// Mitsubishi GX Works2 project: Group29   PLC: FX3G

// global labels: Global1
VAR_GLOBAL
  emergency AT X005 : BOOL;
  low_stock AT M2 : BOOL;
  light7 AT Y007 : BOOL;
  start_work_day AT X007 : BOOL;
  switch1 AT X001 : BOOL;
  inputAnalog AT D8280 : INT;
  outputAnalog AT D1400 : REAL;
END_VAR
VAR_GLOBAL CONSTANT
  const400 : REAL := 400;
  const5 : REAL := 5;
END_VAR
VAR_GLOBAL
  lightPinuk AT M5 : BOOL;
  lightRegular AT M7 : BOOL;
  input_raspberry AT D1100 : REAL;
  raspberry_stock AT D1200 : REAL;
  input_lemon AT D1103 : REAL;
  lemon_stock AT D1203 : REAL;
  input_stabilizer AT D1106 : REAL;
  stabilizer_stock AT D1206 : REAL;
  input_gummies AT D1109 : REAL;
  gummy_stock AT D1209 : REAL;
END_VAR
VAR_GLOBAL CONSTANT
  packages_start : REAL;
END_VAR
VAR_GLOBAL
  packges_regular AT D1212 : REAL;
  low_stock_stop AT M2 : BOOL;
  switchPinuk AT M5 : BOOL;
END_VAR
VAR_GLOBAL CONSTANT
  const6 : REAL := 6;
END_VAR
VAR_GLOBAL
  switchRegular AT M7 : BOOL;
  notInRange AT M9 : BOOL;
  switchNotInRange AT M9 : BOOL;
END_VAR
VAR_GLOBAL CONSTANT
  constantAmountRasperry1 : REAL := 385;
  constantAmountLemon1 : REAL := 665;
  constantAmountStabilzer1 : REAL := 210;
  constantAmountGummy1 : REAL := 70;
END_VAR
VAR_GLOBAL
  enoughRaspberry1 AT M20 : BOOL;
  enoughLemon1 AT M23 : BOOL;
  enoughStabilizer1 AT M26 : BOOL;
  emnoghGummy AT M29 : BOOL;
  emnoghGummy1 AT M29 : BOOL;
END_VAR
VAR_GLOBAL CONSTANT
  constantAmountRasperry2 : REAL := 280;
  constantAmountLemon2 : REAL := 455;
  constantAmountStabilzer2 : REAL := 105;
  constantAmountGummy2 : REAL := 28;
END_VAR
VAR_GLOBAL
  enoughRaspberry2 AT M32 : BOOL;
  enoughLemon2 AT M35 : BOOL;
  enoughStabilizer2 AT M38 : BOOL;
  emnoghGummy2 AT M41 : BOOL;
  fullStock AT M44 : BOOL;
  switchFullStock AT M44 : BOOL;
  lightLowStock AT M2 : BOOL;
  packges_pinuk AT D1215 : REAL;
END_VAR
VAR_GLOBAL CONSTANT
  conatant1 : REAL := 1.0;
END_VAR
VAR_GLOBAL
  Light5Sec AT M70 : BOOL;
  TStimer50 AT TS50 : BOOL;
  Timer5sec AT TC50 : BOOL;
  switch5Sec AT M70 : BOOL;
  switch2 AT X002 : BOOL;
  TStimer80 AT TS80 : BOOL;
  switch3 AT X003 : BOOL;
  LightCooling AT M73 : BOOL;
  switchCooling AT M73 : BOOL;
END_VAR
VAR_GLOBAL CONSTANT
  const80 : REAL := 80;
  const100 : REAL := 100;
  const50 : REAL := 50;
  const70 : REAL := 70;
END_VAR
VAR_GLOBAL
  Timer50 AT TC50 : BOOL;
END_VAR
VAR_GLOBAL CONSTANT
  timer50TV : INT := 50;
END_VAR
VAR_GLOBAL
  Timer80 AT TC80 : BOOL;
END_VAR
VAR_GLOBAL CONSTANT
  timer80TV : INT := 80;
END_VAR
VAR_GLOBAL
  switch7 AT Y007 : BOOL;
  raspberry_cooling_regular AT D1220 : REAL;
  lemon_cooling_regular AT D1223 : REAL;
  raspberry_cooling_pinuk AT D1226 : REAL;
  lemon_cooling_pinuk AT D1229 : REAL;
  Light0 AT Y000 : BOOL;
  Light2 AT Y002 : BOOL;
  raspberry_cooling AT D1226 : REAL;
  lemon_cooling AT D1229 : REAL;
  total_add_raspberry AT D1232 : REAL;
  total_add_lemon AT D1235 : REAL;
  switch0 AT Y000 : BOOL;
  switchMix AT M86 : BOOL;
  mixHelp AT M76 : BOOL;
  Timer5 AT TC5 : BOOL;
END_VAR
VAR_GLOBAL CONSTANT
  const20 : INT := 1;
  const1timer : INT := 1;
END_VAR
VAR_GLOBAL
  TStimer5 AT TS5 : BOOL;
END_VAR
VAR_GLOBAL CONSTANT
  const10timer : INT := 5;
END_VAR
VAR_GLOBAL
  Light5 AT Y005 : BOOL;
  Timer6 AT TC6 : BOOL;
  TStimer6 AT TS6 : BOOL;
  Light6 AT Y006 : BOOL;
  switch5 AT Y005 : BOOL;
  switch6 AT Y006 : BOOL;
  regularCounter AT CC3 : BOOL;
END_VAR
VAR_GLOBAL CONSTANT
  const3 : INT := 3;
END_VAR
VAR_GLOBAL
  outConterRegular AT CS3 : BOOL;
  storage AT D1240 : REAL;
END_VAR
VAR_GLOBAL CONSTANT
  const0 : REAL;
END_VAR
VAR_GLOBAL
  isPinuk AT M79 : BOOL;
  isRegular AT M82 : BOOL;
  LightMix AT M86 : BOOL;
  switchFinishCooling AT Y002 : BOOL;
  light2TurnedOff AT M98 : BOOL;
  MixTimerPinuk AT TC1 : BOOL;
  MixTimerregular AT TC2 : BOOL;
END_VAR
VAR_GLOBAL CONSTANT
  PinukMixDuration : INT := 50;
  RegularMixDuration : INT := 30;
END_VAR
VAR_GLOBAL
  TSRegular AT TS2 : BOOL;
  TSPinuk AT TS1 : BOOL;
END_VAR
VAR_GLOBAL CONSTANT
  const1time5 : INT := 1;
  const5timer : INT := 5;
END_VAR
VAR_GLOBAL
  finishCooling AT M99 : BOOL;
  mAor AT M90 : BOOL;
  finishMix AT M96 : BOOL;
  LightStartMix AT M86 : BOOL;
  switchStartMix AT M86 : BOOL;
  storage_out AT D1280 : REAL;
END_VAR
VAR_GLOBAL CONSTANT
  const40 : REAL := 40;
END_VAR
VAR_GLOBAL
  OUTPUT AT D8282 : DINT;
END_VAR
VAR_GLOBAL CONSTANT
  const350 : REAL := 350;
  const560 : REAL := 560;
  const700 : REAL := 700;
  const490 : REAL := 490;
END_VAR
VAR_GLOBAL
  total_respberry_lemon_pinuk AT D1260 : REAL;
  total_ice_pinuk AT D1260 : REAL;
  Mixing_container AT D1260 : REAL;
  raspberry_cooling_container AT D1226 : REAL;
  lemon_cooling_container AT D1229 : REAL;
END_VAR

// task Task_01 (event TRUE, interval 0, priority 31): POU_01

PROGRAM POU_01
(* structured ladder/FBD written out as ST: instructions are called as NAME(EN, inputs, outputs); _pN, _eN, _tN stand for wires *)
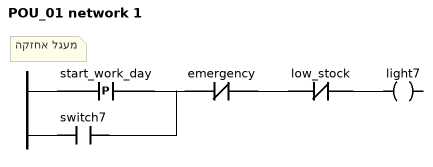
(* network 1 *)
(* מעגל אחזקה *)
light7 := ((LDP(TRUE, start_work_day) OR switch7) AND NOT emergency) AND NOT low_stock;
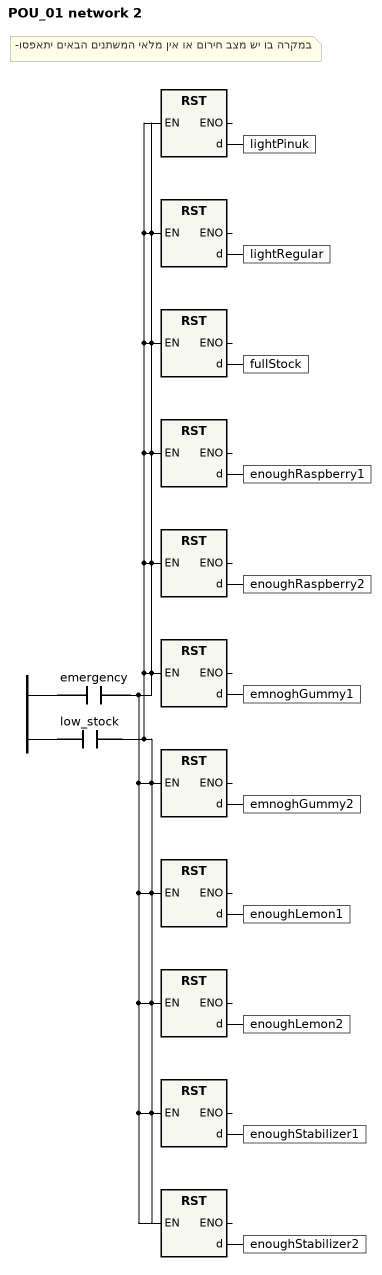
(* network 2 *)
(* במקרה בו יש מצב חירום או אין מלאי המשתנים הבאים יתאפסו- *)
_p1 := emergency OR low_stock;
RST(_p1, lightPinuk);
RST(_p1, lightRegular);
RST(_p1, fullStock);
RST(_p1, enoughRaspberry1);
RST(_p1, enoughRaspberry2);
RST(_p1, emnoghGummy1);
RST(_p1, emnoghGummy2);
RST(_p1, enoughLemon1);
RST(_p1, enoughLemon2);
RST(_p1, enoughStabilizer1);
RST(_p1, enoughStabilizer2);
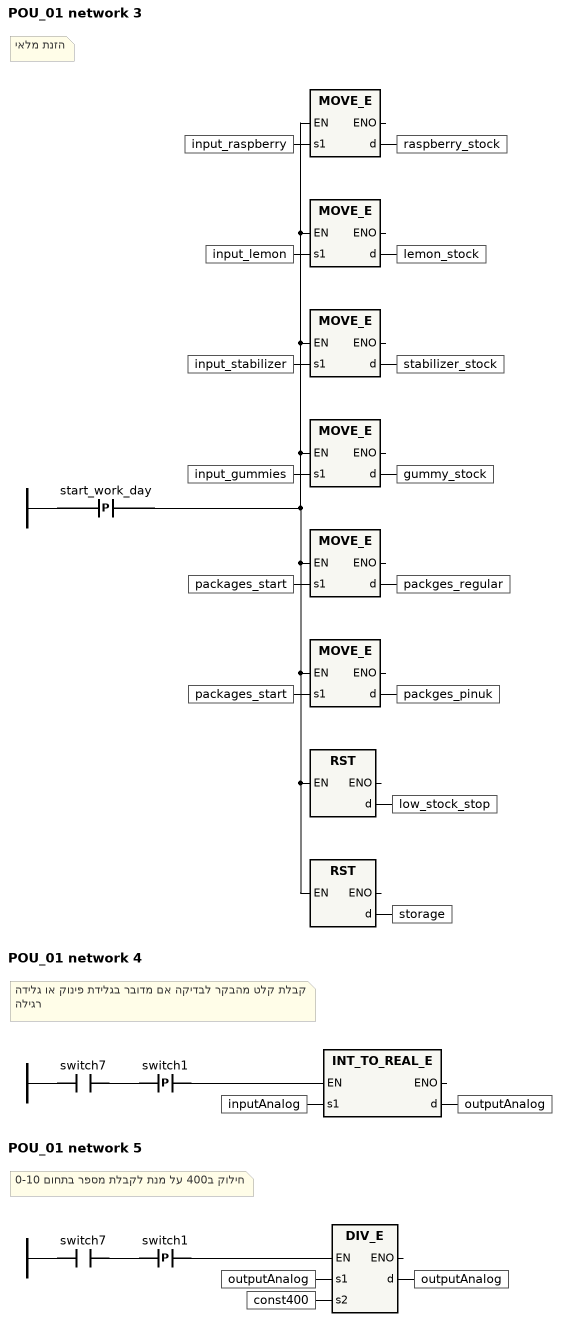
(* network 3 *)
(* הזנת מלאי *)
_p1 := LDP(TRUE, start_work_day);
MOVE_E(_p1, input_raspberry, raspberry_stock);
MOVE_E(_p1, input_lemon, lemon_stock);
MOVE_E(_p1, input_stabilizer, stabilizer_stock);
MOVE_E(_p1, input_gummies, gummy_stock);
MOVE_E(_p1, packages_start, packges_regular);
MOVE_E(_p1, packages_start, packges_pinuk);
RST(_p1, low_stock_stop);
RST(_p1, storage);
(* network 4 *)
(* קבלת קלט מהבקר לבדיקה אם מדובר בגלידת פינוק או גלידה רגילה *)
INT_TO_REAL_E(switch7 AND LDP(TRUE, switch1), inputAnalog, outputAnalog);
(* network 5 *)
(* חילוק ב400 על מנת לקבלת מספר בתחום 0-10 *)
DIV_E(switch7 AND LDP(TRUE, switch1), outputAnalog, const400, outputAnalog);
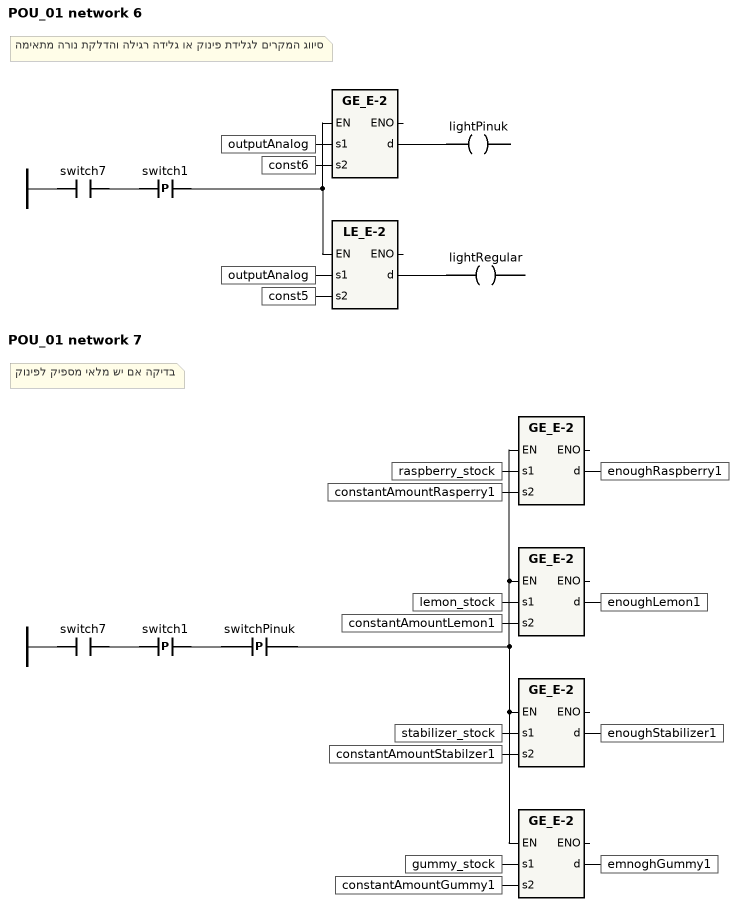
(* network 6 *)
(* סיווג המקרים לגלידת פינוק או גלידה רגילה והדלקת נורה מתאימה *)
_p1 := switch7 AND LDP(TRUE, switch1);
GE_E(_p1, outputAnalog, const6, _t2);
lightPinuk := _t2;
LE_E(_p1, outputAnalog, const5, _t3);
lightRegular := _t3;
(* network 7 *)
(* בדיקה אם יש מלאי מספיק לפינוק *)
_p1 := switch7 AND LDP(TRUE, switch1) AND LDP(TRUE, switchPinuk);
GE_E(_p1, raspberry_stock, constantAmountRasperry1, enoughRaspberry1);
GE_E(_p1, lemon_stock, constantAmountLemon1, enoughLemon1);
GE_E(_p1, stabilizer_stock, constantAmountStabilzer1, enoughStabilizer1);
GE_E(_p1, gummy_stock, constantAmountGummy1, emnoghGummy1);
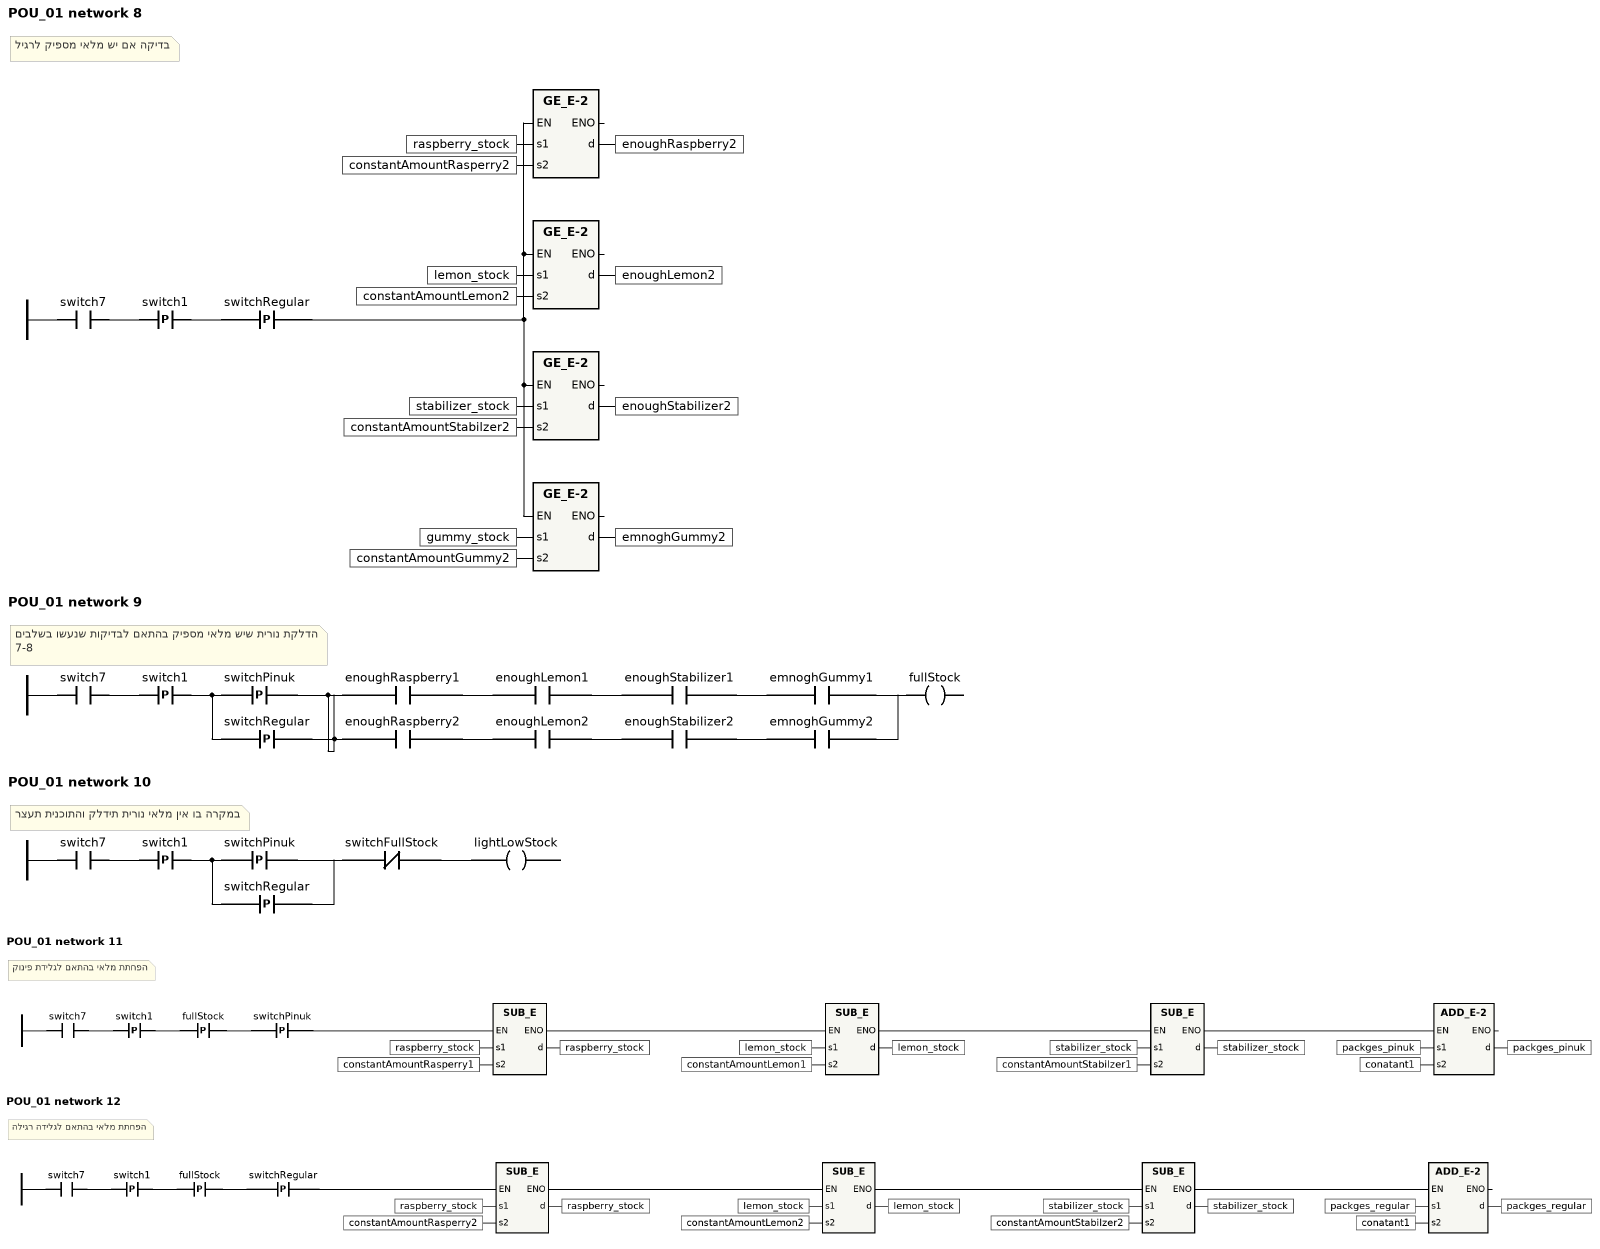
(* network 8 *)
(* בדיקה אם יש מלאי מספיק לרגיל *)
_p1 := switch7 AND LDP(TRUE, switch1) AND LDP(TRUE, switchRegular);
GE_E(_p1, raspberry_stock, constantAmountRasperry2, enoughRaspberry2);
GE_E(_p1, lemon_stock, constantAmountLemon2, enoughLemon2);
GE_E(_p1, stabilizer_stock, constantAmountStabilzer2, enoughStabilizer2);
GE_E(_p1, gummy_stock, constantAmountGummy2, emnoghGummy2);
(* network 9 *)
(* הדלקת נורית שיש מלאי מספיק בהתאם לבדיקות שנעשו בשלבים 7-8 *)
_p1 := switch7 AND LDP(TRUE, switch1);
_p2 := (_p1 AND LDP(TRUE, switchPinuk)) OR (_p1 AND LDP(TRUE, switchRegular));
fullStock := (_p2 AND enoughRaspberry1 AND enoughLemon1 AND enoughStabilizer1 AND emnoghGummy1) OR (_p2 AND enoughRaspberry2 AND enoughLemon2 AND enoughStabilizer2 AND emnoghGummy2);
(* network 10 *)
(* במקרה בו אין מלאי נורית תידלק והתוכנית תעצר *)
_p1 := switch7 AND LDP(TRUE, switch1);
lightLowStock := ((_p1 AND LDP(TRUE, switchPinuk)) OR (_p1 AND LDP(TRUE, switchRegular))) AND NOT switchFullStock;
(* network 11 *)
(* הפחתת מלאי בהתאם לגלידת פינוק *)
_e1 := SUB_E(switch7 AND LDP(TRUE, switch1) AND LDP(TRUE, fullStock) AND LDP(TRUE, switchPinuk), raspberry_stock, constantAmountRasperry1, raspberry_stock);
_e2 := SUB_E(_e1, lemon_stock, constantAmountLemon1, lemon_stock);
_e3 := SUB_E(_e2, stabilizer_stock, constantAmountStabilzer1, stabilizer_stock);
ADD_E(_e3, packges_pinuk, conatant1, packges_pinuk);
(* network 12 *)
(* הפחתת מלאי בהתאם לגלידה רגילה *)
_e1 := SUB_E(switch7 AND LDP(TRUE, switch1) AND LDP(TRUE, fullStock) AND LDP(TRUE, switchRegular), raspberry_stock, constantAmountRasperry2, raspberry_stock);
_e2 := SUB_E(_e1, lemon_stock, constantAmountLemon2, lemon_stock);
_e3 := SUB_E(_e2, stabilizer_stock, constantAmountStabilzer2, stabilizer_stock);
ADD_E(_e3, packges_regular, conatant1, packges_regular);
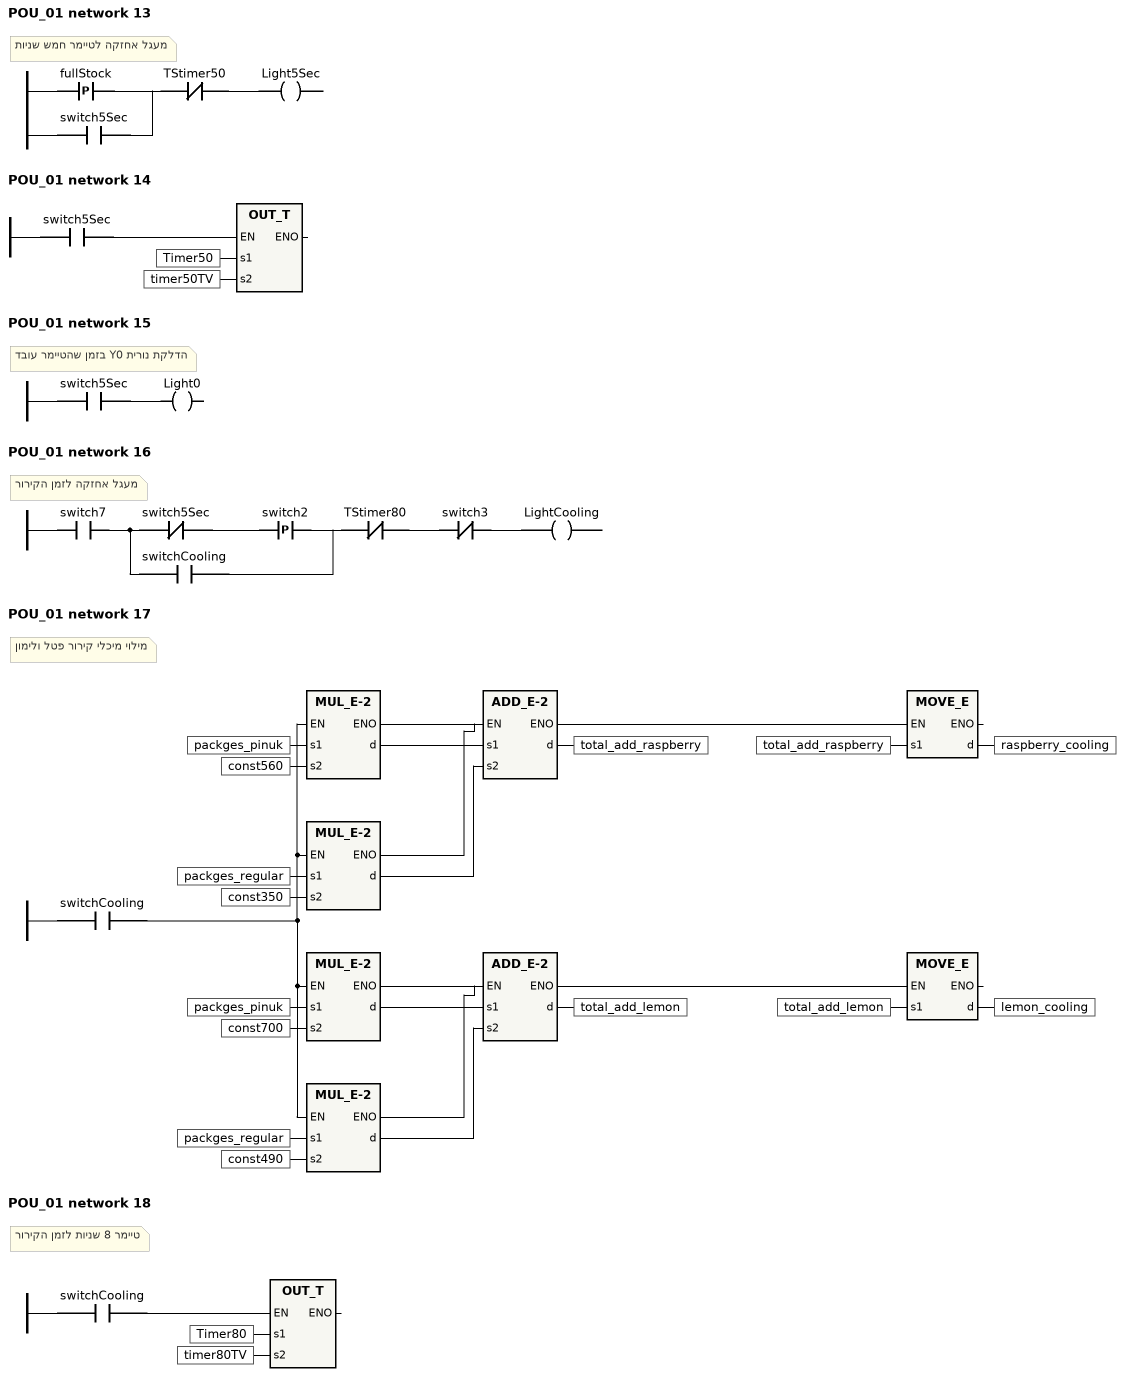
(* network 13 *)
(* מעגל אחזקה לטיימר חמש שניות *)
Light5Sec := (LDP(TRUE, fullStock) OR switch5Sec) AND NOT TStimer50;
(* network 14 *)
OUT_T(switch5Sec, Timer50, timer50TV);
(* network 15 *)
(* הדלקת נורית Y0 בזמן שהטיימר עובד *)
Light0 := switch5Sec;
(* network 16 *)
(* מעגל אחזקה לזמן הקירור *)
LightCooling := (((switch7 AND NOT switch5Sec AND LDP(TRUE, switch2)) OR (switch7 AND switchCooling)) AND NOT TStimer80) AND NOT switch3;
(* network 17 *)
(* מילוי מיכלי קירור פטל ולימון *)
_e2 := MUL_E(switchCooling, packges_pinuk, const560, _t1);
_e4 := MUL_E(switchCooling, packges_regular, const350, _t3);
_e5 := ADD_E(_e2 OR _e4, _t1, _t3, total_add_raspberry);
MOVE_E(_e5, total_add_raspberry, raspberry_cooling);
_e7 := MUL_E(switchCooling, packges_pinuk, const700, _t6);
_e9 := MUL_E(switchCooling, packges_regular, const490, _t8);
_e10 := ADD_E(_e7 OR _e9, _t6, _t8, total_add_lemon);
MOVE_E(_e10, total_add_lemon, lemon_cooling);
(* network 18 *)
(* טיימר 8 שניות לזמן הקירור *)
OUT_T(switchCooling, Timer80, timer80TV);
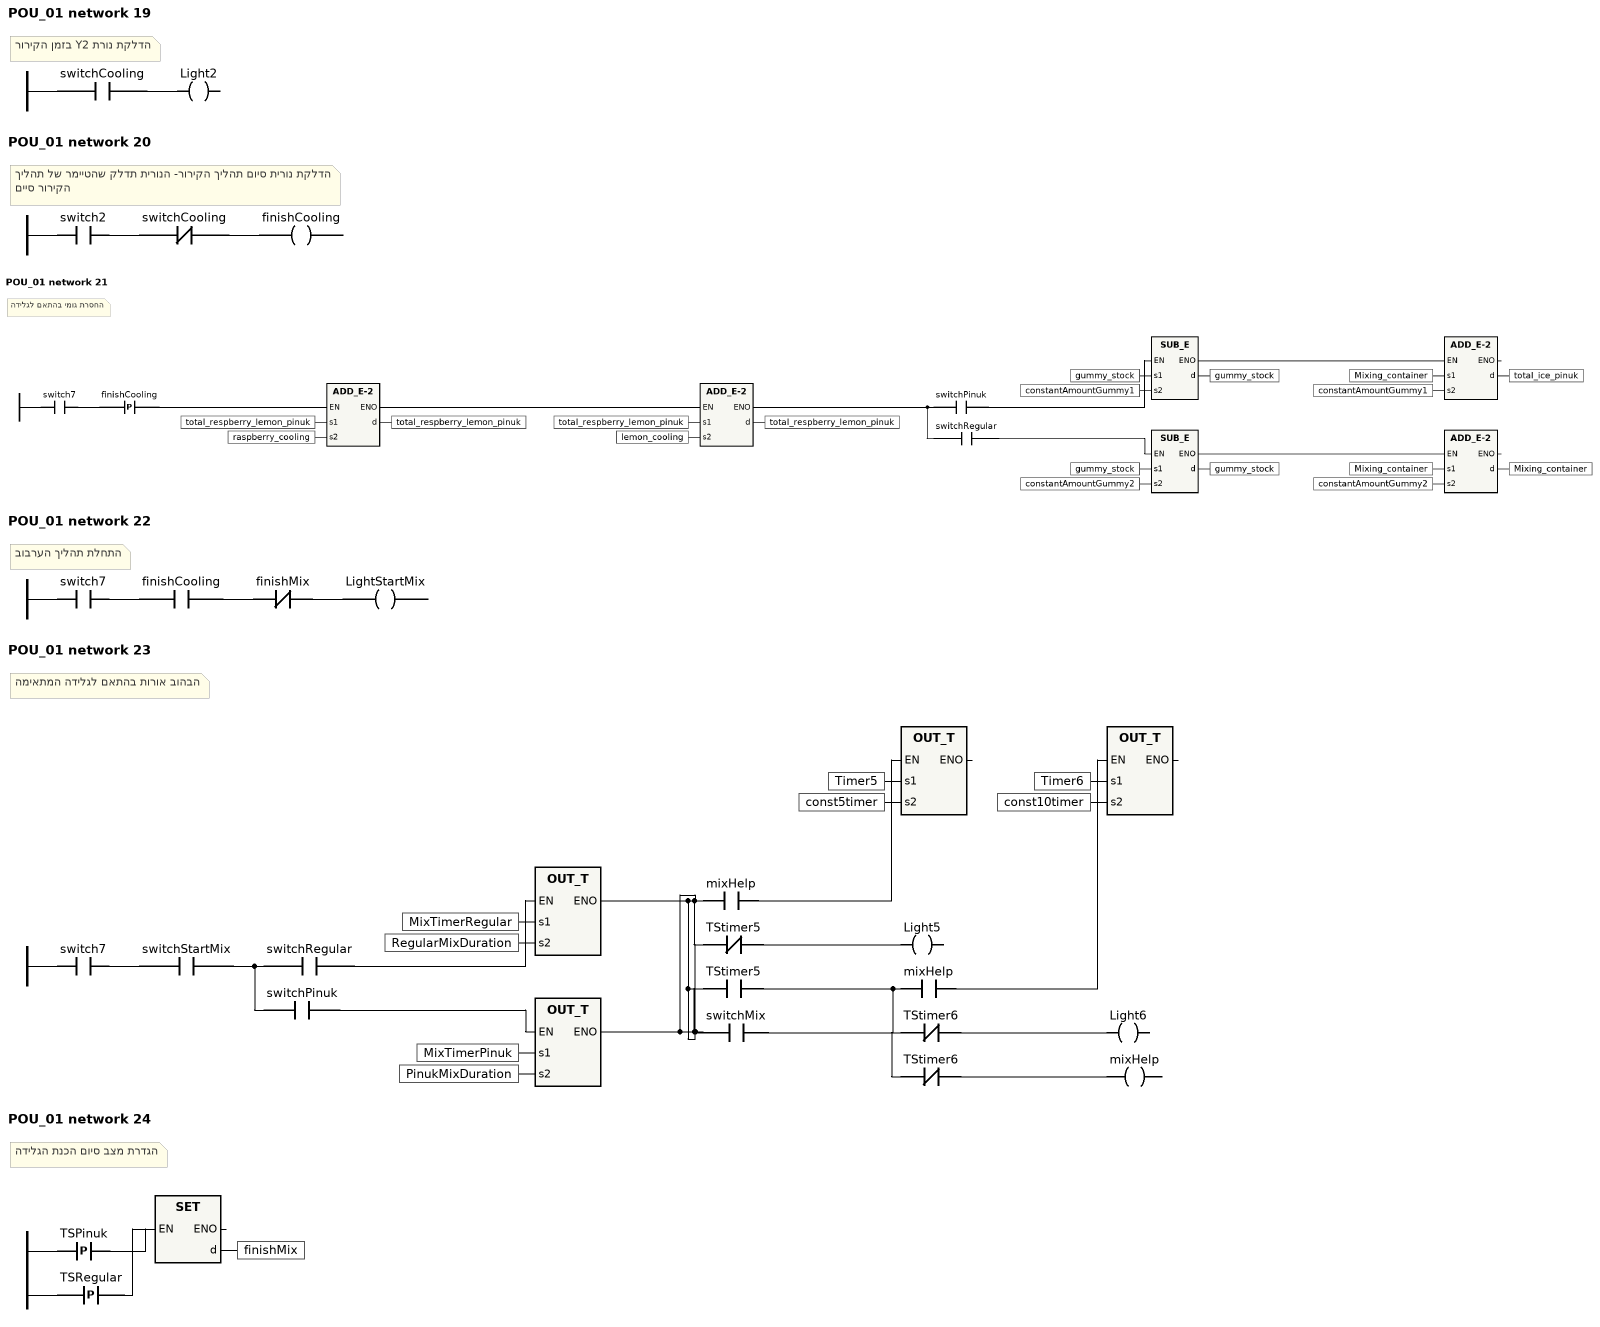
(* network 19 *)
(* הדלקת נורת Y2 בזמן הקירור *)
Light2 := switchCooling;
(* network 20 *)
(* הדלקת נורית סיום תהליך הקירור- הנורית תדלק שהטיימר של תהליך הקירור סיים *)
finishCooling := switch2 AND NOT switchCooling;
(* network 21 *)
(* החסרת גומי בהתאם לגלידה *)
_e1 := ADD_E(switch7 AND LDP(TRUE, finishCooling), total_respberry_lemon_pinuk, raspberry_cooling, total_respberry_lemon_pinuk);
_e2 := ADD_E(_e1, total_respberry_lemon_pinuk, lemon_cooling, total_respberry_lemon_pinuk);
_e3 := SUB_E(_e2 AND switchPinuk, gummy_stock, constantAmountGummy1, gummy_stock);
ADD_E(_e3, Mixing_container, constantAmountGummy1, total_ice_pinuk);
_e4 := SUB_E(_e2 AND switchRegular, gummy_stock, constantAmountGummy2, gummy_stock);
ADD_E(_e4, Mixing_container, constantAmountGummy2, Mixing_container);
(* network 22 *)
(* התחלת תהליך הערבוב *)
LightStartMix := switch7 AND finishCooling AND NOT finishMix;
(* network 23 *)
(* הבהוב אורות בהתאם לגלידה המתאימה *)
_p1 := switch7 AND switchStartMix;
_e2 := OUT_T(_p1 AND switchRegular, MixTimerRegular, RegularMixDuration);
_e3 := OUT_T(_p1 AND switchPinuk, MixTimerPinuk, PinukMixDuration);
_p4 := _e2 OR _e3;
OUT_T(_p4 AND mixHelp, Timer5, const5timer);
Light5 := _p4 AND NOT TStimer5;
_p5 := _p4 AND TStimer5;
OUT_T(_p5 AND mixHelp, Timer6, const10timer);
Light6 := _p5 AND NOT TStimer6;
mixHelp := _p4 AND switchMix AND NOT TStimer6;
(* network 24 *)
(* הגדרת מצב סיום הכנת הגלידה *)
SET(LDP(TRUE, TSPinuk) OR LDP(TRUE, TSRegular), finishMix);
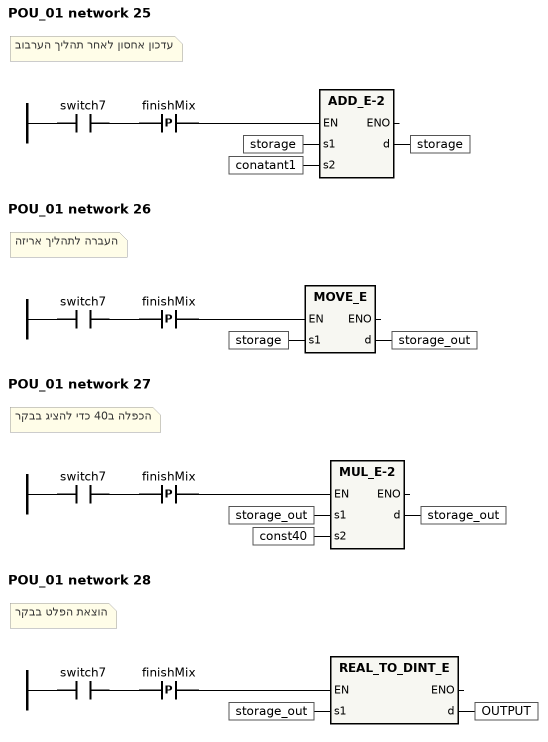
(* network 25 *)
(* עדכון אחסון לאחר תהליך הערבוב *)
ADD_E(switch7 AND LDP(TRUE, finishMix), storage, conatant1, storage);
(* network 26 *)
(* העברה לתהליך אריזה *)
MOVE_E(switch7 AND LDP(TRUE, finishMix), storage, storage_out);
(* network 27 *)
(* הכפלה ב40 כדי להציג בבקר *)
MUL_E(switch7 AND LDP(TRUE, finishMix), storage_out, const40, storage_out);
(* network 28 *)
(* הוצאת הפלט בבקר *)
REAL_TO_DINT_E(switch7 AND LDP(TRUE, finishMix), storage_out, OUTPUT);
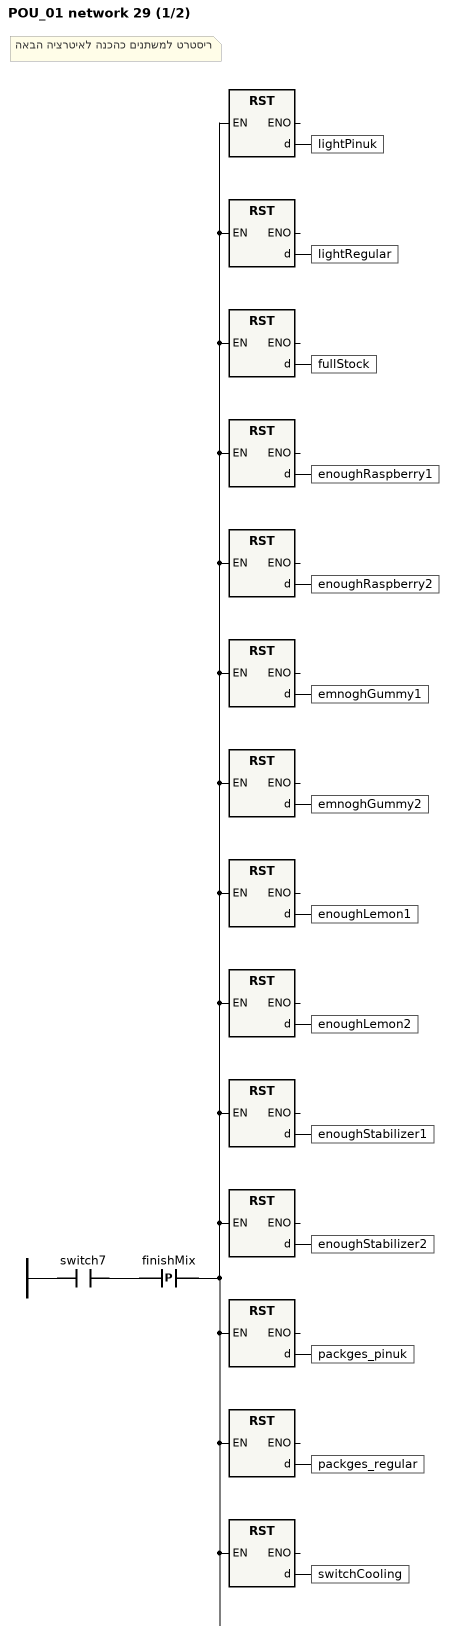
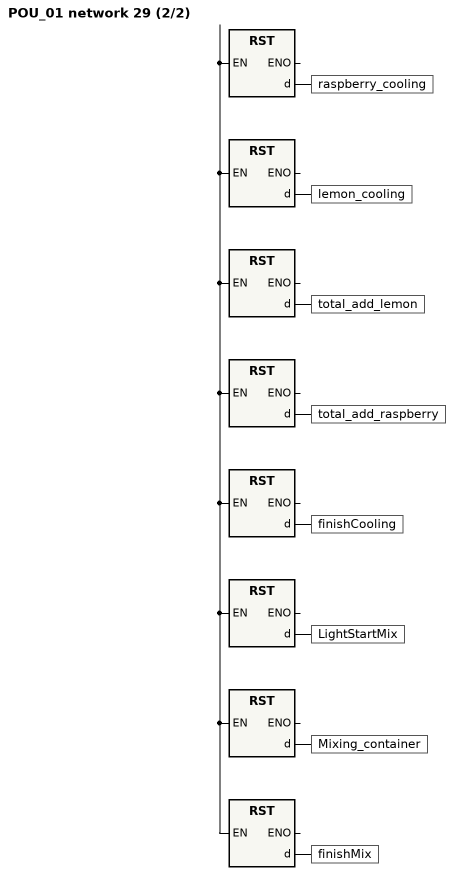
(* network 29 *)
(* ריסטרט למשתנים כהכנה לאיטרציה הבאה *)
_p1 := switch7 AND LDP(TRUE, finishMix);
RST(_p1, lightPinuk);
RST(_p1, lightRegular);
RST(_p1, fullStock);
RST(_p1, enoughRaspberry1);
RST(_p1, enoughRaspberry2);
RST(_p1, emnoghGummy1);
RST(_p1, emnoghGummy2);
RST(_p1, enoughLemon1);
RST(_p1, enoughLemon2);
RST(_p1, enoughStabilizer1);
RST(_p1, enoughStabilizer2);
RST(_p1, packges_pinuk);
RST(_p1, packges_regular);
RST(_p1, switchCooling);
RST(_p1, raspberry_cooling);
RST(_p1, lemon_cooling);
RST(_p1, total_add_lemon);
RST(_p1, total_add_raspberry);
RST(_p1, finishCooling);
RST(_p1, LightStartMix);
RST(_p1, Mixing_container);
RST(_p1, finishMix);
END_PROGRAM
